// TIA Portal V17 export
// export: Created 2022-07-20T07:01:33.5356929Z, ExportSetting WithDefaults, DisplayName Totally Integrated Automation Portal, DisplayVersion V17, DisplayName TIA Portal Openness, DisplayVersion V17, DisplayName TIA Portal Version Control Interface, DisplayVersion V17, DisplayName SINAMICS Startdrive Advanced, DisplayVersion V17, DisplayName SINAMICS Startdrive G130, G150, S120, S150, SINAMICS MV, S210, DisplayVersion V17, DisplayName SINAMICS Startdrive G110M, G120, G120C, G120D, G120P, G115D, DisplayVersion V17, DisplayName STEP 7 Professional, DisplayVersion V17, DisplayName STEP 7 Safety, DisplayVersion V17, DisplayName WinCC Advanced, DisplayVersion V17
FUNCTION_BLOCK "FB10320_PrinterHeatingManifoldManager"   // FB10320, LAD
{ S7_Optimized_Access := 'TRUE' }
VERSION : 0.1
// stored: AutoNumber false, IsIECCheckEnabled false, IsRetainMemResEnabled false, MemoryReserve 100, SetENOAutomatically false, UDAEnableTagReadback false
   VAR_INPUT
      ManifoldTemperatureRawValue : Int;
      ManifoldTemperatureSetPoint : Real;
      RequestHeatManifold : Bool;
      RequestResetManifoldInError : Bool;
   END_VAR
   VAR_OUTPUT
      ActiveHeatingManifold : Bool;
      ManifoldActualTemperature : Real;
      ManifoldHeatingInProgress : Bool;
      ManifoldInError : Bool;
      ManifoldOverheating : Bool;
   END_VAR
   VAR
      ManifoldStateDiagram : Int;
      TON_ManifoldHeatingSafety : TON_TIME;
      R_TRIG_RequestHeatingManifold { S7_SetPoint := 'True'} : R_TRIG;
      F_TRIG_RequesHeatingManifold { S7_SetPoint := 'True'} : F_TRIG;
      ManifoldLowLimitTemperature { S7_SetPoint := 'True'} : Real;
      ManifoldHighLimitTemperature : Real;
   END_VAR
   VAR CONSTANT
      WAIT_FOR_HEATING_MANIFOLD_REQUEST : Int := 0;
      HEATING_MANIFOLD_IN_PROGRESS : Int := 10;
      HEATING_MANIFOLD_SETPOINT_REACHED : Int := 20;
      HEATING_MANIFOLD_DELTA_LOW_LIMIT : Real := 2.0;
      HEATING_MANIFOLD_DELTA_HIGH_LIMIT : Real := 10.0;
   END_VAR
BEGIN

REGION Network 1 (SCL): First Scan
   IF "FirstScan" THEN
       #ActiveHeatingManifold := FALSE;
       #ManifoldActualTemperature := 0.0;
       #ManifoldHeatingInProgress := FALSE;
       #ManifoldInError := FALSE;
       #ManifoldOverheating := FALSE;
       #ManifoldStateDiagram := #WAIT_FOR_HEATING_MANIFOLD_REQUEST;
       #ManifoldLowLimitTemperature := #ManifoldTemperatureSetPoint - #HEATING_MANIFOLD_DELTA_LOW_LIMIT;
       #ManifoldHighLimitTemperature := #ManifoldTemperatureSetPoint + #HEATING_MANIFOLD_DELTA_HIGH_LIMIT;
   END_IF;
END_REGION

REGION Network 2 (SCL): Edge Signals & Timers
   REGION EDGE SIGNALS
       #R_TRIG_RequestHeatingManifold(CLK := #RequestHeatManifold);
   END_REGION

   REGION TIMERS
       #TON_ManifoldHeatingSafety(IN := #ManifoldHeatingInProgress,
                                  PT := T#200s);
   END_REGION
END_REGION

REGION Network 3 (SCL): Heating Manifold Management
   CASE #ManifoldStateDiagram OF

       #WAIT_FOR_HEATING_MANIFOLD_REQUEST: //STATE 0
           IF  #R_TRIG_RequestHeatingManifold.Q THEN
               #ManifoldStateDiagram := #HEATING_MANIFOLD_IN_PROGRESS;
           END_IF;
           #ManifoldHeatingInProgress := FALSE;
           #ActiveHeatingManifold := FALSE;

       #HEATING_MANIFOLD_IN_PROGRESS: //STATE 1
           IF #ManifoldActualTemperature >= #ManifoldTemperatureSetPoint THEN
               #ManifoldStateDiagram := #HEATING_MANIFOLD_SETPOINT_REACHED;
           END_IF;
           #ManifoldHeatingInProgress := TRUE;
           #ActiveHeatingManifold := TRUE;

       #HEATING_MANIFOLD_SETPOINT_REACHED: //STATE 2
           IF #ManifoldActualTemperature <= #ManifoldLowLimitTemperature THEN
               #ManifoldStateDiagram := #HEATING_MANIFOLD_IN_PROGRESS;
           END_IF;
           #ActiveHeatingManifold := FALSE;

   END_CASE;


   IF NOT (#RequestHeatManifold) THEN
       #ManifoldStateDiagram := #WAIT_FOR_HEATING_MANIFOLD_REQUEST;
   END_IF;
END_REGION

REGION Network 4 (SCL): Manifold Error Management
   IF #TON_ManifoldHeatingSafety.Q THEN
       #ManifoldInError := TRUE;
   END_IF;

   IF #RequestResetManifoldInError THEN
       #ManifoldInError := FALSE;
   END_IF;

   #ManifoldOverheating := #ManifoldActualTemperature > #ManifoldHighLimitTemperature;

   IF #ManifoldInError OR #ManifoldOverheating THEN
       #ManifoldStateDiagram := #WAIT_FOR_HEATING_MANIFOLD_REQUEST;
   END_IF;
END_REGION

REGION Network 5 (SCL)
   ///!\\\
   //MODIFIER VALEUR AVEC VALEUR REELLE DU CAPTEUR
   //!\\
   "FC10020_Linearization"(X1 := 0,
                           Y1 := 0,
                           X2 := 24576.0,
                           Y2 := 150,
                           X := #ManifoldTemperatureRawValue,
                           Y => #ManifoldActualTemperature);
END_REGION
END_FUNCTION_BLOCK
